TYPE "ValveConfig"
VERSION : 0.1
// Block: ValveConfig
   STRUCT
      RestLimSwitchExist : Bool;
      WorkLimSwitchExist : Bool;
      CheckOilInPressure : Bool;
      CutRestWhenIsAtRest : Bool;
      CutWorkWhenIsAtWork : Bool;
      RestTime : Time;
      WorkTime : Time;
      RestTimeOut : Time;
      WorkTimeOut : Time;
   END_STRUCT;

END_TYPE
